# EPICS alarm handler configuration: alh_files/mgnt_in20Dl.alhConfig
GROUP NULL MGNT:IN20DL:1
   $COMMAND edm -x -eolc -noedit mgnt_in20_main.edl

$ALIAS IN20DL
$GUIDANCE
in20 Dog Leg Region
   Group Name: MGNT:IN20DL:1
   Summary PV:  MGNT:IN20DL:1:STATSUMY
$END

   INCLUDE MGNT:IN20DL:1 ./mgnt_in20Dl_bend.alhConfig
   INCLUDE MGNT:IN20DL:1 ./mgnt_in20Dl_lgps.alhConfig
   INCLUDE MGNT:IN20DL:1 ./mgnt_in20Dl_quad.alhConfig
   INCLUDE MGNT:IN20DL:1 ./mgnt_in20Dl_xcor.alhConfig
   INCLUDE MGNT:IN20DL:1 ./mgnt_in20Dl_ycor.alhConfig
